FUNCTION_BLOCK ABSTRACT CommunicationSettings
VAR_INPUT
	DefaultOperationTimeout : TIME := Tc2_System.DEFAULT_ADS_TIMEOUT;
END_VAR

PROPERTY ABSTRACT CommunicationTypeName : STRING
GET
END_GET
END_PROPERTY

END_FUNCTION_BLOCK

(* stored: Version 1.1.0.1
   POU CommunicationSettings: Id {e05e7971-f90f-4e84-a2e2-8680d10b5b1e}, SpecialFunc None
   Property CommunicationTypeName: Id {55c07768-0d4b-4381-b100-780dd7a23e81}
   Get Get: Id {948df464-6698-47f0-b35b-261586637032} *)
